{attribute addProperty BoxType "EL2912-0000-0016"}
{attribute addProperty Id "FSoE_CommandUSINT811FSOUT_Module_1_OutputBIT10.1251FSOUT_Module_1_ErrAckBIT10.1251FSOUT_Module_2_OutputBIT10.1251FSOUT_Module_2_ErrAckBIT10.1251FSoE_CRC_000UINT1623FSoE_Connection_IDUINT1622"}
{attribute addProperty CRC "978345874"}
{attribute addProperty SizeInBites "48"}
{attribute addProperty SizeInBytes "6"}
TYPE FSOE_3A505F92 :
STRUCT
	{attribute addProperty Name "FSoE_Command"}
	FSoE_Command : USINT;
	{attribute addProperty Name "FSOUT_Module_1_Output"}
	FSOUT_Module_1_Output : BIT;
	{attribute addProperty Name "FSOUT_Module_1_ErrAck"}
	FSOUT_Module_1_ErrAck : BIT;
	{attribute addProperty Name "FSOUT_Module_2_Output"}
	FSOUT_Module_2_Output : BIT;
	{attribute addProperty Name "FSOUT_Module_2_ErrAck"}
	FSOUT_Module_2_ErrAck : BIT;
	{attribute 'hide'}
	reserve_1_BIT_0 : BIT;
	{attribute 'hide'}
	reserve_1_BIT_1 : BIT;
	{attribute 'hide'}
	reserve_1_BIT_2 : BIT;
	{attribute 'hide'}
	reserve_1_BIT_3 : BIT;
	{attribute addProperty Name "FSoE_CRC_000"}
	FSoE_CRC_000 : UINT;
	{attribute addProperty Name "FSoE_Connection_ID"}
	FSoE_Connection_ID : UINT;
END_STRUCT
END_TYPE

(* stored: Version 1.2.0.0, ProductVersion 3.1.4024.9
   DUT FSOE_3A505F92: Id {68823b10-05a9-48b4-b361-4f26dacfb3bd} *)
